# EPICS autosave request: iocBoot/iocUSBC9513/auto_settings.req
#file "C9513_settings.req", P=C9513:
#file "1608G_settings.req", P=1608G:
file "USBCTR_settings.req", P=USBCTR:
